(* IEC 61131-3 sources: std_i2980_v2.06_cp053/Source/IMM/ieccontrol/AutoCalibration1 (part 5) *)

@F

@Trans @RT(9)TResetBwd @F @T @F @F @T @T @TL(2)
TRUE

@RT(9)TResetBwd @F
@Goto @RT(7)S_RESET @F @F

@Step @RT(23)S_CHECK_ALARMS_RETRYBWD @F @F @F @F @RT(0) @F
@AcbCont @RT(7)unnamed @F 0

@AltBranch @RT(3)alt @F 2
@TransSeq @RT(4)tseq @F 1
@Trans @RT(9)TRetryBwd @F @T @F @F @T @T @TL(2)
S_CHECK_ALARMS_RETRYBWD.T > T#1s

@RT(9)TRetryBwd @F

@TransSeq @RT(4)tseq @F 2
@Trans @RT(14)TStopIdentBwd4 @F @T @F @F @T @F @TL(2)
sv_iPendingAlarms <> 0

@RT(14)TStopIdentBwd4 @F
@Goto @RT(13)S_StopMoveFwd @F @F

@Goto @RT(11)S_CALIB_BWD @F @F

@Step @RT(12)S_MoveEndBwd @F @F @F @F @RT(0) @F
@AcbCont @RT(7)unnamed @F 3
@Acb @RT(11)AMoveEndBwd @F @T @RT(1)P @RT(0) @F @F @T @TL(27)
bMoveBwdDone := FALSE;

IF mActMovement^.bPositionIncreasingFwd THEN
   mActMovement^.prIdentPosition^ := mrBwdStopPosition;
ELSE
   mActMovement^.prIdentPosition^ := mActMovement^.prStroke^ - mrBwdStopPosition;
END_IF;
mActMovement^.prStopRamp^ := 1.0e10;
mActMovement^.pConstBwdVis^.Pressure.Output.rRamp := MAX(1.0e20,mActMovement^.pConstBwdVis^.Pressure.Output.rRamp);
mActMovement^.pConstBwdVis^.Pressure.rMinOutput := 0.1 * rMaxPressureLimit;
sv_EjectorIdentMinMovement.pConstBwdVis^.Pressure.Output.rRamp := MAX(1.0e10, sv_EjectorIdentMinMovement.pConstBwdVis^.Pressure.Output.rRamp);
sv_EjectorIdentMinMovement.pConstBwdVis^.Pressure.rMinOutput := 0.1 * sv_EjectorIdentMinMovement.prMaxPressureBwd^;

mActMovement^.pbMoveIdent^ := TRUE;

evStartRequestData.DeviceId := mActMovement^.DeviceId;
evStartRequestData.MoveDir := cMoveBwd;
IF mActMovement^.MoveId > cMoveNone THEN
   evStartRequestData.MoveId := cMoveDecompAftPlast;
ELSE
   evStartRequestData.MoveId := cMoveBwd;
END_IF;
miErrorNo := cIdentSpeedMaxEnd;

SET_EVENT(evStartRequest, evStartRequestData);

@F
@Acb @RT(21)ACheckMoveEndBwdReady @F @T @RT(1)N @RT(0) @F @F @T @TL(5)
fbCheckReady(DeviceId := evStartRequestData.DeviceId);
IF fbCheckReady.bReady THEN
   bMoveBwdDone := TRUE;
END_IF;

@F
@Acb @RT(16)AMoveEndBwdReady @F @T @RT(2)P0 @RT(0) @F @F @T @TL(2)
aStopMovementBwd();

@F

@AltBranch @RT(3)alt @F 2
@TransSeq @RT(4)tseq @F 1
@Trans @RT(15)TMoveEndBwdDone @F @T @F @F @T @T @TL(2)
bMoveBwdDone

@RT(15)TMoveEndBwdDone @F

@TransSeq @RT(4)tseq @F 4
@Trans @RT(15)TStopMoveEndBwd @F @T @F @F @T @F @TL(4)
sv_GlobalIdentMaxSpeedStatus.Status = tnCalibState_Aborted OR
sv_GlobalIdentMaxSpeedStatus.Status = tnCalibState_None
OR sv_iPendingAlarms <> 0

@RT(15)TStopMoveEndBwd @F
@Step @RT(16)S_StopMoveEndBwd @F @F @F @F @RT(0) @F
@AcbCont @RT(7)unnamed @F 1
@Acb @RT(15)AStopMoveEndBwd @F @T @RT(1)P @RT(0) @F @F @T @TL(2)
aStopMovementError(sMovementName := CONCAT(sMoveName, ' max ident Bwd to end position'));

@F

@Trans @RT(16)TResetMoveEndBwd @F @T @F @F @T @F @TL(2)
TRUE

@RT(16)TResetMoveEndBwd @F
@Goto @RT(7)S_RESET @F @F

@Step @RT(6)S_Done @F @F @F @F @RT(0) @F
@AcbCont @RT(7)unnamed @F 1
@Acb @RT(5)ADone @F @T @RT(1)P @RT(0) @F @F @T @TL(6)
mActMovement^.Status := tnCalibState_Done;
sv_GlobalIdentMaxSpeedStatus.Status := tnCalibState_Done;

mActMovement^.prVelocityFwd^ := rSpeedLimitFwd;
mActMovement^.prVelocityBwd^ := rSpeedLimitBwd;

@F

@Trans @RT(5)TDone @F @T @F @F @T @T @TL(2)
TRUE

@RT(5)TDone @F
@Goto @RT(7)S_RESET @F @F
@END_SfcData
@SaActions 0
@SaTrans 0
@SaExits 0
@END_SfcBody

@@@BEG_Comment@@@
@TL(0)

@@@END_Comment@@@

@BEG_Body
@TL(35)
//stop all calibrations
// TEST
IF sv_GlobalIdentMaxSpeedStatus.Command = tnCalibCommand_Stop THEN
    sv_GlobalIdentMaxSpeedStatus.bStart := FALSE;
END_IF;
//
IF sv_GlobalIdentMaxSpeedStatus.Command = tnCalibCommand_Stop OR (NOT sv_GlobalIdentMaxSpeedStatus.bStart) THEN
    FOR i:= 1 TO cCalibMovements DO
        IF CHECK_REF(sv_GlobalIdentMaxSpeedStatus.pMovements[i]^) THEN
            IF sv_GlobalIdentMaxSpeedStatus.pMovements[i]^.Status = tnCalibState_Running OR
               sv_GlobalIdentMaxSpeedStatus.pMovements[i]^.bRedo THEN
                sv_GlobalIdentMaxSpeedStatus.pMovements[i]^.Status := tnCalibState_Aborted;
                sv_GlobalIdentMaxSpeedStatus.pMovements[i]^.bRedo := FALSE;//FIXME: check if needed
                sv_GlobalIdentMaxSpeedStatus.Status := tnCalibState_Aborted;
                EXIT;
            END_IF;
        END_IF;
    END_FOR;
    IF (sv_GlobalIdentMaxSpeedStatus.Command = tnCalibCommand_Stop) THEN
       IF (sv_GlobalIdentMaxSpeedStatus.Status <> tnCalibState_Aborted) THEN
          sv_GlobalIdentMaxSpeedStatus.Status := tnCalibState_None;
       END_IF;

    END_IF;
ELSIF (sv_GlobalIdentMaxSpeedStatus.Command = tnCalibCommand_Start) OR (sv_GlobalIdentMaxSpeedStatus.bStart) THEN
    IF sv_OperationMode = nSetup THEN
        mbUseSingleMovement := FALSE;
        START_PROCESS_ALGORITHM(paMaxCalibSequence);
    ELSE
        sv_GlobalIdentMaxSpeedStatus.bStart := FALSE;
        SET_ALARM(erSetupModeRequiredForCalib);
    END_IF;
END_IF;
sv_GlobalIdentMaxSpeedStatus.Command := tnCalibCommand_None;

@END_Body

@@@BEG_Comment@@@
@TL(0)

@@@END_Comment@@@

@BEG_SfcBody
18 18 17

@BEG_SfcData 2
@StepSeq @RT(4)sseq @F 15
@Step @RT(7)S_RESET @F @F @T @F @RT(0) @F
@AcbCont @RT(7)unnamed @F 3
@Acb @RT(6)AReset @F @T @RT(1)P @RT(0) @F @F @T @TL(2)
sv_bAutoIdentRunning := FALSE;

@F
@Acb @RT(14)AStopMovements @F @T @RT(1)N @RT(0) @F @F @T @TL(12)
(* stop all identification movements *)
FOR i:= 1 TO cCalibMovements DO
    IF CHECK_REF(sv_GlobalIdentMaxSpeedStatus.pMovements[i]^) THEN
        IF sv_GlobalIdentMaxSpeedStatus.pMovements[i]^.Status = tnCalibState_Running OR
           sv_GlobalIdentMaxSpeedStatus.pMovements[i]^.bRedo THEN
            sv_GlobalIdentMaxSpeedStatus.pMovements[i]^.Status := tnCalibState_Aborted;
            sv_GlobalIdentMaxSpeedStatus.pMovements[i]^.bRedo := FALSE;//FIXME: check if needed
            EXIT;
        END_IF;
    END_IF;
END_FOR;

@F
@Acb @RT(9)AStopSelf @F @T @RT(1)P @RT(0) @F @F @T @TL(3)
sv_GlobalIdentMaxSpeedStatus.bStart := FALSE;
STOP_PROCESS_ALGORITHM();

@F

@Trans @RT(7)Trans50 @F @T @F @F @T @T @TL(2)
TRUE

@RT(7)Trans50 @F
@Step @RT(6)S_INIT @F @T @F @F @RT(0) @F
@AcbCont @RT(7)unnamed @F 2
@Acb @RT(11)ASortCalibs @F @T @RT(1)P @RT(0) @F @F @T @TL(24)
sv_GlobalIdentMaxSpeedStatus.Status := tnCalibState_Running;
miErrorNo := 0;

tmpMovements := sv_GlobalIdentMaxSpeedStatus.pMovements;

(* get number of movements *)
FOR i:= 1 TO cCalibMovements DO
    IF NOT CHECK_REF(tmpMovements[i]^)  THEN
        EXIT;
    END_IF;
END_FOR;
iMaxMovements := i -1;

(* sort them by iOrder *)
FOR i := 1 TO iMaxMovements -1 DO
    FOR j := 1 TO iMaxMovements - 1 - i +1 DO
        IF tmpMovements[j]^.iOrder > tmpMovements[j + 1]^.iOrder THEN
            tmpM := tmpMovements[j];
            tmpMovements[j] := tmpMovements[j + 1];
            tmpMovements[j + 1] := tmpM;
        END_IF;
    END_FOR;
END_FOR;

@F
@Acb @RT(9)Action108 @F @T @RT(1)P @RT(0) @F @F @T @TL(3)
mCalibCounter := 0;
sv_GlobalIdentMaxSpeedStatus.iCurrentStep := mCalibCounter;

@F

@AltBranch @RT(3)alt @F 2
@TransSeq @RT(4)tseq @F 1
@Trans @RT(7)Trans80 @F @T @F @F @T @T @TL(3)
NOT sv_bCoresActive AND
sv_iPendingAlarms = 0

@RT(7)Trans80 @T @TL(5)
Comment : Start with moving ejector and
mold in backward position, check if any failure
occured.
After that start the calibration cycle, if no alarm is
pending

@TransSeq @RT(4)tseq @F 4
@Trans @RT(7)Trans87 @F @T @F @F @T @F @TL(3)
sv_bCoresActive OR
sv_iPendingAlarms > 0

@RT(7)Trans87 @F
@Step @RT(6)Step74 @F @F @F @F @RT(0) @F
@AcbCont @RT(7)unnamed @F 1
@Acb @RT(14)AAnyCoreActive @F @F @RT(1)N @RT(0) @F @F @F @F

@Trans @RT(7)Trans88 @F @T @F @F @T @T @TL(3)
TRUE

@RT(7)Trans88 @F
@Goto @RT(7)S_RESET @F @F

@Step @RT(6)Step19 @F @F @F @F @RT(0) @F
@AcbCont @RT(7)unnamed @F 1
@Acb @RT(12)ASignalStart @F @T @RT(1)P @RT(0) @F @F @T @TL(2)
sv_bAutoIdentRunning := TRUE;

@F

@Trans @RT(7)Trans18 @F @T @F @F @T @T @TL(2)
TRUE

@RT(7)Trans18 @F
@Step @RT(17)S_MoveEjectorBack @F @F @F @F @RT(0) @F
@AcbCont @RT(7)unnamed @F 3
@Acb @RT(12)AEjectorBack @F @F @RT(1)P @RT(0) @F @F @F @F
@Acb @RT(9)Action116 @F @T @RT(1)N @RT(0) @F @F @T @TL(2)
fbCheckReady(DeviceId := DeviceIdEjector)

@F
@Acb @RT(17)AResetEjectorBack @F @T @RT(2)P0 @RT(0) @F @F @T @TL(7)
miErrorNo := 0;
sv_EjectorIdentMaxMovement.prIdentPosition^ := 0.0;
sv_EjectorIdentMaxMovement.prStopRamp^ := 0.0;
sv_EjectorIdentMaxMovement.pbMoveIdent^ := FALSE;
sv_EjectorIdentMaxMovement.pConstBwdVis^ := ConstBwdVis;

@F

@AltBranch @RT(3)alt @F 2
@TransSeq @RT(4)tseq @F 1
@Trans @RT(7)Trans72 @F @T @F @F @T @T @TL(3)
fbCheckReady.bReady AND
sv_iPendingAlarms = 0

@RT(7)Trans72 @F

@TransSeq @RT(4)tseq @F 4
@Trans @RT(7)Trans83 @F @T @F @F @T @F @TL(4)
sv_GlobalIdentMaxSpeedStatus.Status = tnCalibState_Aborted OR
sv_GlobalIdentMaxSpeedStatus.Status = tnCalibState_None
OR sv_iPendingAlarms <> 0

@RT(7)Trans83 @F
@Step @RT(13)S_StopEjector @F @F @F @F @RT(0) @F
@AcbCont @RT(7)unnamed @F 1
@Acb @RT(16)AStopEjeMovement @F @F @RT(1)P @RT(0) @F @F @F @F

@Trans @RT(7)Trans84 @F @T @F @F @T @T @TL(3)
TRUE

@RT(7)Trans84 @F
@Goto @RT(7)S_RESET @F @F

@Step @RT(14)S_MoveMoldBack @F @F @F @F @RT(0) @F
@AcbCont @RT(7)unnamed @F 3
@Acb @RT(9)AMoldBack @F @F @RT(1)P @RT(0) @F @F @F @F
@Acb @RT(9)Action118 @F @T @RT(1)N @RT(0) @F @F @T @TL(2)
fbCheckReady(DeviceId := DeviceIdMold)

@F
@Acb @RT(14)AResetMoldBack @F @T @RT(2)P0 @RT(0) @F @F @T @TL(7)
miErrorNo := 0;
sv_MoldIdentMaxMovement.prIdentPosition^ := 0.0;
sv_MoldIdentMaxMovement.prStopRamp^ := 0.0;
sv_MoldIdentMaxMovement.pbMoveIdent^ := FALSE;
sv_MoldIdentMaxMovement.pConstBwdVis^ := ConstBwdVis;

@F

@AltBranch @RT(3)alt @F 2
@TransSeq @RT(4)tseq @F 1
@Trans @RT(7)Trans81 @F @T @F @F @T @T @TL(3)
fbCheckReady.bReady AND
sv_iPendingAlarms = 0

@RT(7)Trans81 @F

@TransSeq @RT(4)tseq @F 4
@Trans @RT(7)Trans85 @F @T @F @F @T @F @TL(4)
sv_GlobalIdentMaxSpeedStatus.Status = tnCalibState_Aborted OR
sv_GlobalIdentMaxSpeedStatus.Status = tnCalibState_None
OR sv_iPendingAlarms <> 0

@RT(7)Trans85 @F
@Step @RT(10)S_StopMold @F @F @F @F @RT(0) @F
@AcbCont @RT(7)unnamed @F 1
@Acb @RT(17)AStopMoldMovement @F @F @RT(1)P @RT(0) @F @F @F @F

@Trans @RT(7)Trans86 @F @T @F @F @T @T @TL(2)
TRUE

@RT(7)Trans86 @F
@Goto @RT(7)S_RESET @F @F

@Step @RT(14)S_CALIB_SINGLE @F @F @T @F @RT(0) @F
@AcbCont @RT(7)unnamed @F 1
@Acb @RT(19)AStartMovementStart @F @T @RT(1)P @RT(0) @F @F @T @TL(5)
IF mCalibCounter < iMaxMovements THEN
   mCalibCounter := mCalibCounter +1;
   tmpMovements[mCalibCounter]^.bRedo := TRUE;
END_IF;

@F

@AltBranch @RT(3)alt @F 2
@TransSeq @RT(4)tseq @F 1
@Trans @RT(18)TCheckActMoveReady @F @T @F @F @T @T @TL(4)
tmpMovements[mCalibCounter]^.bRedo = FALSE AND
NOT(sv_GlobalIdentMaxSpeedStatus.Status = tnCalibState_Aborted OR
    sv_GlobalIdentMaxSpeedStatus.Status = tnCalibState_Error)

@RT(18)TCheckActMoveReady @F

@TransSeq @RT(4)tseq @F 2
@Trans @RT(11)TCheckError @F @T @F @F @T @F @TL(4)
sv_GlobalIdentMaxSpeedStatus.Status = tnCalibState_Aborted OR
sv_GlobalIdentMaxSpeedStatus.Status = tnCalibState_Error OR
iMaxMovements = 0

@RT(11)TCheckError @F
@Goto @RT(7)S_RESET @F @F

@Step @RT(11)S_CHECKNEXT @F @F @F @F @RT(0) @F
@AcbCont @RT(7)unnamed @F 0

@AltBranch @RT(3)alt @F 2
@TransSeq @RT(4)tseq @F 1
@Trans @RT(9)TNextUnit @F @T @F @F @T @T @TL(2)
mCalibCounter < iMaxMovements

@RT(9)TNextUnit @F

@TransSeq @RT(4)tseq @F 4
@Trans @RT(10)TStopIdent @F @T @F @F @T @T @TL(2)
mCalibCounter >= iMaxMovements

@RT(10)TStopIdent @F
@Step @RT(11)S_StopIdent @F @F @F @F @RT(0) @F
@AcbCont @RT(7)unnamed @F 1
@Acb @RT(10)AStopIdent @F @T @RT(1)P @RT(0) @F @F @T @TL(2)
sv_GlobalIdentMaxSpeedStatus.Status := tnCalibState_Done;

@F

@Trans @RT(6)TReset @F @T @F @F @T @T @TL(2)
TRUE

@RT(6)TReset @F
@Goto @RT(7)S_RESET @F @F

@Goto @RT(14)S_CALIB_SINGLE @F @F
@END_SfcData
@SaActions 5
@SaText @RT(12)AEjectorBack 1 @TL(20)
miErrorNo := cIdentSpeedMaxSequence;

IF sv_EjectorIdentMaxMovement.bPositionIncreasingFwd THEN
   sv_EjectorIdentMaxMovement.prIdentPosition^ := mrBwdStopPosition;
ELSE
   sv_EjectorIdentMaxMovement.prIdentPosition^ := sv_EjectorIdentMaxMovement.prStroke^ - mrBwdStopPosition;
END_IF;
sv_EjectorIdentMaxMovement.prStopRamp^ := 1.0e10;
ConstBwdVis := sv_EjectorIdentMaxMovement.pConstBwdVis^;
sv_EjectorIdentMaxMovement.pConstBwdVis^.Pressure.Output.rRamp := MAX(1.0e10, sv_EjectorIdentMaxMovement.pConstBwdVis^.Pressure.Output.rRamp);
sv_EjectorIdentMaxMovement.pConstBwdVis^.Pressure.rMinOutput := 0.1 * sv_EjectorIdentMaxMovement.prMaxPressureBwd^;
sv_EjectorIdentMaxMovement.pbMoveIdent^ := TRUE;

evStartRequestData.DeviceId := DeviceIdEjector;
evStartRequestData.MoveDir := cMoveBwd;
evStartRequestData.MoveId := cMoveBwd;
SET_EVENT(evStartRequest, evStartRequestData);

@SaText @RT(9)AMoldBack 1 @TL(19)
miErrorNo := cIdentSpeedMaxSequence;

IF sv_MoldIdentMaxMovement.bPositionIncreasingFwd THEN
   sv_MoldIdentMaxMovement.prIdentPosition^ := mrBwdStopPosition;
ELSE
   sv_MoldIdentMaxMovement.prIdentPosition^ := sv_MoldIdentMaxMovement.prStroke^ - mrBwdStopPosition;
END_IF;
sv_MoldIdentMaxMovement.prStopRamp^ := 1.0e10;
ConstBwdVis := sv_MoldIdentMaxMovement.pConstBwdVis^;
sv_MoldIdentMaxMovement.pConstBwdVis^.Pressure.Output.rRamp := MAX(1.0e10, sv_MoldIdentMaxMovement.pConstBwdVis^.Pressure.Output.rRamp);
sv_MoldIdentMaxMovement.pConstBwdVis^.Pressure.rMinOutput := 0.1 * sv_MoldIdentMaxMovement.prMaxPressureBwd^;
sv_MoldIdentMaxMovement.pbMoveIdent^ := TRUE;

evStartRequestData.DeviceId := DeviceIdMold;
evStartRequestData.MoveDir := cMoveBwd;
evStartRequestData.MoveId := cMoveBwd;
SET_EVENT(evStartRequest, evStartRequestData);

@SaText @RT(16)AStopEjeMovement 1 @TL(9)
evStopRequestData.DeviceId := DeviceIdEjector;
evStopRequestData.MoveDir := cMoveBwd;
evStopRequestData.MoveId := cMoveBwd;
SET_EVENT(evStopRequest, evStopRequestData);
IF sv_GlobalIdentMaxSpeedStatus.Status <> tnCalibState_None THEN
    sv_GlobalIdentMaxSpeedStatus.Status := tnCalibState_Aborted;
END_IF;

@SaText @RT(17)AStopMoldMovement 1 @TL(9)
evStopRequestData.DeviceId := DeviceIdMold;
evStopRequestData.MoveDir := cMoveBwd;
evStopRequestData.MoveId := cMoveBwd;
SET_EVENT(evStopRequest, evStopRequestData);
IF sv_GlobalIdentMaxSpeedStatus.Status <> tnCalibState_None THEN
    sv_GlobalIdentMaxSpeedStatus.Status := tnCalibState_Aborted;
END_IF;

@SaText @RT(14)AAnyCoreActive 1 @TL(6)
IF sv_bCoresActive THEN
   SET_ALARM(erCalibCoresActive);
END_IF;
sv_GlobalIdentMaxSpeedStatus.Status := tnCalibState_Aborted;

@SaTrans 0
@SaExits 1
@SaExit @SaText @RT(14)E_NotSetupMode 1 @TL(2)
sv_OperationMode <> nSetup

@RT(7)S_RESET @RT(1)1 @F @F @SaSfc @RT(14)E_NotSetupMode 5 @RT(5)DUMMY
@BEG_SfcData 2
@ExitSeq @RT(4)sseq @F 3
@Step @RT(8)unnamed1 @F @T @F @F @RT(0) @F
@AcbCont @RT(7)unnamed @F 0

@Trans @RT(8)unnamed3 @F @T @F @F @T @T @TL(2)

@RT(8)unnamed3 @F
@Goto @RT(9)unlabeled @F @F
@END_SfcData

@END_SfcBody

@@@BEG_Comment@@@
@TL(2)
Coordinate sequential start of auto calib cycle
starts one auto calib movement after the other
@@@END_Comment@@@

@BEG_Body
@TL(7)
IF (rStep > 0.0) THEN
   rRealValue := (0.999 + rActNumber / rStep);
   rRoundedNumber := DINT_TO_REAL(TRUNC_TO_DINT(rRealValue)) * rStep;
ELSE
   rRoundedNumber := rActNumber;
END_IF;

@END_Body

@@@BEG_Comment@@@
@TL(0)

@@@END_Comment@@@

@BEG_Body
@TL(39)
IF bStart THEN
   rMaxRefSpeed := rMaxSpeedLimit;
   rMinRefSpeed := 0.0;
END_IF;
IF (bUnstable OR bTimeOut) THEN
   // increase speed
   IF (rActRefSpeed >= rMFactorMaxMinLimit * rMaxSpeedLimit) THEN
      bMinDetected := TRUE;
      rMinSpeed := rActRefSpeed;
      RETURN;
   END_IF;
   rMinRefSpeed := rActRefSpeed;
   bMinDetected := FALSE;
  IF (rMaxRefSpeed - rMinRefSpeed) < (0.0025 * rMaxSpeedLimit) THEN
  // difference to low to maximum - stop or increase maximum?
      bMinDetected := TRUE;
      rMinSpeed := rMaxRefSpeed;
   ELSIF (rMaxRefSpeed < rMaxSpeedLimit) AND (rMinRefSpeed > 0.0) THEN
      rRefSpeed := 0.5 * (rMaxRefSpeed + rMinRefSpeed);
      bMinDetected := FALSE;
   ELSE
      rRefSpeed := rActRefSpeed + 0.01 * rMaxSpeedLimit;
      IF (rRefSpeed >= rMaxSpeedLimit) THEN
         bMinDetected := TRUE;
         rMinSpeed := rMaxSpeedLimit;
      END_IF;
   END_IF;
ELSE
   // reduce speed
   rMaxRefSpeed := rActRefSpeed;
   IF (rMaxRefSpeed - rMinRefSpeed) < (0.0025 * rMaxSpeedLimit) THEN
      bMinDetected := TRUE;
      rMinSpeed := rActRefSpeed;
   ELSE
      bMinDetected := FALSE;
      rRefSpeed := 0.5 * (rMaxRefSpeed + rMinRefSpeed);
   END_IF;
END_IF;

@END_Body

@@@BEG_Comment@@@
@TL(0)

@@@END_Comment@@@

@BEG_Body
@TL(26)
bIdentActive := FALSE;
FOR i:= 1 TO cCalibMovements DO
   IF CHECK_REF(sv_GlobalIdentMinSpeedStatus.pMovements[i]^) THEN
      IF sv_GlobalIdentMinSpeedStatus.pMovements[i]^.bRedo THEN
         mActMovement := sv_GlobalIdentMinSpeedStatus.pMovements[i];
         bIdentActive := TRUE;
         sv_GlobalIdentMinSpeedStatus.iCurrentStep :=  i;
         mCalibCounter := i;
         IF sv_OperationMode = nSetup THEN
            mbUseSingleMovement := TRUE;
            START_PROCESS_ALGORITHM(paMinSingleMovement);
         ELSE
            sv_GlobalIdentMinSpeedStatus.pMovements[i]^.bRedo := FALSE;
            SET_ALARM(erSetupModeRequiredForCalib);
         END_IF;
         EXIT;
      END_IF;
   END_IF;
END_FOR;
IF ((NOT bIdentActive) AND (sv_GlobalIdentMinSpeedStatus.Status = tnCalibState_Running)) THEN
   sv_GlobalIdentMinSpeedStatus.Status := tnCalibState_Done;
END_IF;

STOP_PROCESS_ALGORITHM();

@END_Body

@@@BEG_Comment@@@
@TL(0)

@@@END_Comment@@@

@BEG_Body
@TL(4)

START_PROCESS_ALGORITHM(paRedoMin);

@END_Body

@@@BEG_Comment@@@
@TL(0)

@@@END_Comment@@@

@BEG_SfcBody
44 51 50

@BEG_SfcData 2
@StepSeq @RT(4)sseq @F 39
@Step @RT(7)S_RESET @F @F @T @F @RT(0) @F
@AcbCont @RT(7)unnamed @F 0

@Trans @RT(7)Trans47 @F @T @F @F @T @T @TL(2)
mbLogFileSaved

@RT(7)Trans47 @F
@Step @RT(6)S_STOP @F @F @F @F @RT(0) @F
@AcbCont @RT(7)unnamed @F 1
@Acb @RT(9)AStopSelf @F @T @RT(1)P @RT(0) @F @F @T @TL(18)
IF (sv_GlobalIdentMinSpeedStatus.Status = tnCalibState_Aborted) THEN
   mActMovement^.prVelocityFwd^ := rSpeedLimitFwd;
   mActMovement^.prVelocityBwd^ := rSpeedLimitBwd;
END_IF;
sv_GlobalIdentMinSpeedStatus.Command := tnCalibCommand_None;
sv_bAutoIdentRunning := FALSE;
mActMovement^.bRedo := FALSE;
mActMovement^.pdMaxMoveTimeFwd^ := dMaxMoveTimeSaveFwd;
mActMovement^.pdMaxMoveTimeBwd^ := dMaxMoveTimeSaveBwd;
mActMovement^.prStopRamp^ := 0.0;
mActMovement^.pConstFwdVis^ := ConstVisFwd;
mActMovement^.pConstBwdVis^ := ConstVisBwd;

//release memory
abSpeedMeasure.aEnd();

STOP_PROCESS_ALGORITHM();

@F

@Trans @RT(8)TRestart @F @T @F @F @T @T @TL(2)
TRUE

@RT(8)TRestart @F
@Step @RT(6)S_INIT @F @T @F @F @RT(0) @F
@AcbCont @RT(7)unnamed @F 1
@Acb @RT(7)Action3 @F @T @RT(1)P @RT(0) @F @F @T @TL(38)
miErrorNo := 0;

sv_GlobalIdentMinSpeedStatus.Status := tnCalibState_Running;
mActMovement^.Status := tnCalibState_Running;
sMoveName := mActMovement^.sName;

abSpeedMeasure.aInit();

bMinFwdRetry := FALSE;
bMinBwdRetry := FALSE;

dMaxMoveTimeSaveFwd := mActMovement^.pdMaxMoveTimeFwd^;
dMaxMoveTimeSaveBwd := mActMovement^.pdMaxMoveTimeBwd^;

ConstVisFwd := mActMovement^.pConstFwdVis^;
ConstVisBwd := mActMovement^.pConstBwdVis^;

rSpeedLimitFwd := mActMovement^.prVelocityFwd^;
rSpeedLimitBwd := mActMovement^.prVelocityBwd^;

IF (mActMovement^.rMaxPositionLimitFactor > mActMovement^.rMinPositionLimitFactor) AND
   (mActMovement^.rMinPositionLimitFactor > 0.0) AND (mActMovement^.rMaxPositionLimitFactor < 1.0) THEN
   mrMaxPositionFactor := mActMovement^.rMaxPositionLimitFactor;
   mrMinPositionFactor := mActMovement^.rMinPositionLimitFactor;
ELSE // use deafult values
   mrMaxPositionFactor := 0.8;
   mrMinPositionFactor := 0.2;
END_IF;

rMaxPressureFwd := 0.0;
rMaxPressureBwd := 0.0;
mprActPressure := sv_PumpData[mActMovement^.DeviceId.IndexId].prActSysPressure;
IF CHECK_REF(mprActPressure^) THEN
   mbprActPressureLinked := TRUE;
ELSE
   mbprActPressureLinked := FALSE;
END_IF;

@F

@Trans @RT(13)TMoveStartBwd @F @T @F @F @T @T @TL(3)
TRUE

@RT(13)TMoveStartBwd @F
@Step @RT(14)S_MoveStartBwd @F @F @F @F @RT(0) @F
@AcbCont @RT(7)unnamed @F 3
@Acb @RT(13)AMoveStartBwd @F @T @RT(1)P @RT(0) @F @F @T @TL(4)
bMoveBwdDone := FALSE;
miErrorNo := cIdentSpeedMinBwdInit;
aStartMovementBwd();

@F
@Acb @RT(23)ACheckMoveStartBwdReady @F @T @RT(1)N @RT(0) @F @F @T @TL(5)
fbCheckReady(DeviceId := evStartRequestData.DeviceId);
IF fbCheckReady.bReady THEN
   bMoveBwdDone := TRUE;
END_IF;

@F
@Acb @RT(18)AMoveStartBwdReady @F @T @RT(2)P0 @RT(0) @F @F @T @TL(5)
aStopMovementBwd();

@F

@AltBranch @RT(3)alt @F 2
@TransSeq @RT(4)tseq @F 1
@Trans @RT(8)TInitBwd @F @T @F @F @T @T @TL(2)
bMoveBwdDone

@RT(8)TInitBwd @F

@TransSeq @RT(4)tseq @F 4
@Trans @RT(17)TStopMoveStartBwd @F @T @F @F @T @F @TL(5)
sv_GlobalIdentMinSpeedStatus.Status = tnCalibState_Aborted OR
sv_GlobalIdentMinSpeedStatus.Status = tnCalibState_None
OR sv_iPendingAlarms <> 0
OR mActMovement^.bRedo = FALSE

@RT(17)TStopMoveStartBwd @F
@Step @RT(18)S_StopMoveStartBwd @F @F @T @F @RT(0) @F
@AcbCont @RT(7)unnamed @F 1
@Acb @RT(22)AStopMoveErrorStartBwd @F @T @RT(1)P @RT(0) @F @F @T @TL(2)
aStopMovementError(sMovementName := CONCAT(sMoveName, ' min ident Fwd: Bwd to initial position'));

@F

@Trans @RT(6)TReset @F @T @F @F @T @F @TL(2)
TRUE

@RT(6)TReset @F
@Goto @RT(7)S_RESET @F @F

@Step @RT(22)S_CHECK_ALARMS_INITBWD @F @F @F @F @RT(0) @F
@AcbCont @RT(7)unnamed @F 0

@AltBranch @RT(3)alt @F 2
@TransSeq @RT(4)tseq @F 1
@Trans @RT(11)TStartIdent @F @T @F @F @T @T @TL(2)
S_CHECK_ALARMS_INITBWD.T > T#100ms

@RT(11)TStartIdent @F

@TransSeq @RT(4)tseq @F 2
@Trans @RT(12)TStopInitBwd @F @T @F @F @T @F @TL(2)
sv_iPendingAlarms <> 0

@RT(12)TStopInitBwd @F
@Goto @RT(18)S_StopMoveStartBwd @F @F

@Step @RT(15)S_INITCALIB_FWD @F @F @F @F @RT(0) @F
@AcbCont @RT(7)unnamed @F 1
@Acb @RT(13)aInitIdentFwd @F @T @RT(1)P @RT(0) @F @F @T @TL(26)
iFileCounter := 1;
IF (CHECK_REF(mActMovement^.prSizeFactorFwd^)) THEN
   IF (mActMovement^.prSizeFactorFwd^ > 0.0) THEN
      rVelocitSizeFactor := mActMovement^.prSizeFactorFwd^;
   END_IF;
ELSE
   rVelocitSizeFactor := 1.0;
END_IF;
rRefSpeedLimit := 0.01 * mActMovement^.prVelocityLimitFwd^;
rMaxPressureLimit := mActMovement^.prMaxPressureFwd^;
IF CHECK_REF(mActMovement^.prMaxPressureFwdHydr^) THEN
   rMaxRefPressureLimit := mActMovement^.prMaxPressureFwdHydr^;
   IF (rMaxRefPressureLimit > 0.0) THEN
      rPressureFactorFwd := rMaxPressureLimit / rMaxRefPressureLimit;
   ELSE
      rPressureFactorFwd := 1.0;
   END_IF;
ELSE
   rMaxRefPressureLimit := mActMovement^.prMaxPressureFwd^;
   rPressureFactorFwd := 1.0;
END_IF;

aCalcMinSpeedOutput.bStart := TRUE;

dummy := Print('Calib min output %s Fwd started', sMoveName);

@F

@Trans @RT(7)TDelay1 @F @T @F @F @T @T @TL(2)
S_INITCALIB_FWD.T>T#100ms

@RT(7)TDelay1 @F
@Step @RT(11)S_CALIB_FWD @F @F @T @F @RT(0) @F
@AcbCont @RT(7)unnamed @F 4
@Acb @RT(8)ADoCalib @F @T @RT(1)P @RT(0) @F @F @T @TL(67)
// save actual settings
mActMovement^.pConstFwdVis^.Velocity.Output.rOutputValue := rRefSpeedLimit * rVelocitSizeFactor;
mActMovement^.pConstFwdVis^.Velocity.rMinOutput := 0.0;
mActMovement^.pConstFwdVis^.Pressure.Output.rOutputValue := MAX(mActMovement^.pConstFwdVis^.Pressure.Output.rOutputValue, rMaxPressureLimit);
mActMovement^.pConstFwdVis^.Pressure.Output.rRamp := MAX(1.0e10, ConstVisFwd.Pressure.Output.rRamp);
IF mActMovement^.bPositionIncreasingFwd THEN
   mActMovement^.prIdentPosition^ := mActMovement^.prStroke^ * mrMaxPositionFactor;
   mrMinLimitPosition := rStartFactor * mActMovement^.prIdentPosition^ + (1.0 - rStartFactor) * mActMovement^.prPosition^;
   IF (mActMovement^.prIdentPosition^ - mActMovement^.prPosition^) > 0.0 THEN
      rMinStopRamp := rMinStrokeFactor * rRefSpeedLimit  * rRefSpeedLimit / ABS(mActMovement^.prIdentPosition^ - mActMovement^.prPosition^);
   ELSE
      rMinStopRamp := 0.0;
   END_IF;
   mActMovement^.prStopRamp^ := MAX(mActMovement^.pConstFwdVis^.Velocity.Output.rRamp, rMinStopRamp);
   mrMaxLimitPosition := mActMovement^.prIdentPosition^ - 0.5 * rRefSpeedLimit  * rRefSpeedLimit / mActMovement^.prStopRamp^;
ELSE
   mActMovement^.prIdentPosition^ := mActMovement^.prStroke^ * mrMinPositionFactor;
   mrMaxLimitPosition := (1.0 - rStartFactor) * mActMovement^.prPosition^ + rStartFactor * mActMovement^.prIdentPosition^;
   IF (mActMovement^.prPosition^ - mActMovement^.prIdentPosition^) > 0.0 THEN
      rMinStopRamp := rMinStrokeFactor * rRefSpeedLimit  * rRefSpeedLimit / ABS(mActMovement^.prIdentPosition^ - mActMovement^.prPosition^);
   ELSE
      rMinStopRamp := 0.0;
   END_IF;
   mActMovement^.prStopRamp^ := MAX(mActMovement^.pConstFwdVis^.Velocity.Output.rRamp, rMinStopRamp);
   mrMinLimitPosition := mActMovement^.prIdentPosition^ + 0.5 * rRefSpeedLimit  * rRefSpeedLimit / mActMovement^.prStopRamp^;
END_IF;
mActMovement^.pbMoveIdent^ := TRUE;
bMoveIdentDone := FALSE;

bMinFwdDetected := FALSE;

mrRefVelocity := rRefSpeedLimit;
mrRefPressure := rMaxRefPressureLimit;

aStartMeasurement();

bStopUnstable := FALSE;
bTimeOut := FALSE;
IF rRefSpeedLimit > 0.0 THEN
   rMoveStrokeTime := mActMovement^.prStroke^ / rRefSpeedLimit;
ELSE
   rMoveStrokeTime := 0.0;
END_IF;
dMaxMoveTime := T#5s + LINT_TO_TIME(REAL_TO_LINT(rMoveStrokeTime*1.0e6));
IF (dMaxMoveTime > dMoveTimeLimit) THEN
   dMaxMoveTime := dMoveTimeLimit;
   bMoveTimeLimited := TRUE;
   rStartPosition := mActMovement^.prPosition^;
   IF (mActMovement^.bPositionIncreasingFwd) THEN
      rMinMovementPosition := rStartPosition + 0.1 * (mrMaxLimitPosition - mrMinLimitPosition);
   ELSE;
      rMinMovementPosition := rStartPosition - 0.1 * (mrMaxLimitPosition - mrMinLimitPosition );
   END_IF;
ELSE
   bMoveTimeLimited := FALSE;
END_IF;
TimeOut(IN := FALSE,
        PT := dMaxMoveTime);
IF (mActMovement^.pdMaxMoveTimeFwd^ < dMaxMoveTime + dMoveTimeOffset) THEN
   mActMovement^.pdMaxMoveTimeFwd^ := dMaxMoveTime + dMoveTimeOffset;
END_IF;
mActMovement^.prVelocityFwd^ := rRefSpeedLimit;

sWriteSpeedLimit := REAL_TO_STRING(rRefSpeedLimit);
dummy := Print('Calib min output: act. min output: %s', sWriteSpeedLimit);
miErrorNo := cIdentSpeedMinFwdIdent;

@F
@Acb @RT(17)AStartMovementFwd @F @T @RT(1)P @RT(0) @F @F @T @TL(10)
evStartRequestData.DeviceId := mActMovement^.DeviceId;
evStartRequestData.MoveDir := cMoveFwd;
IF mActMovement^.MoveId > cMoveNone THEN
   evStartRequestData.MoveId := mActMovement^.MoveId;
ELSE
   evStartRequestData.MoveId := cMoveFwd;
END_IF;
SET_EVENT(evStartRequest, evStartRequestData);

@F
@Acb @RT(25)ACheckActMovementFwdReady @F @T @RT(1)N @RT(0) @F @F @T @TL(26)
fbCheckReady(DeviceId := evStartRequestData.DeviceId);

TimeOut(IN := TRUE);
IF (fbCheckReady.bReady) THEN
   aStopMeasurement();
   aStopMovementFwd();
   bMoveIdentDone := TRUE;
ELSIF (TimeOut.Q) THEN
   aStopMeasurement();
   aStopMovementFwd();
   IF (bMoveTimeLimited) AND
     ((mActMovement^.bPositionIncreasingFwd AND (mActMovement^.prPosition^ > rMinMovementPosition)) OR
      (NOT mActMovement^.bPositionIncreasingFwd AND (mActMovement^.prPosition^ < rMinMovementPosition))) THEN
      bMoveIdentDone := TRUE;
      dummy := Print('Calib min output: max move time reached with act. min output %s', sWriteSpeedLimit);
   ELSE
      bTimeOut := TRUE;
      dummy := Print('Calib min output: timeout with act. min output %s', sWriteSpeedLimit);
   END_IF;
ELSIF (abSpeedMeasure.aMeasure.bSpeedUnStable) THEN
   aStopMeasurement();
   aStopMovementFwd();
   bStopUnstable := TRUE;
   dummy := Print('Calib min output: unstable speed with act. min output %s', sWriteSpeedLimit);
END_IF;

@F
@Acb @RT(16)AStopMovementFwd @F @T @RT(2)P0 @RT(0) @F @F @T @TL(8)
mActMovement^.prStopRamp^ := 0.0;
mActMovement^.pConstFwdVis^ := ConstVisFwd;
mActMovement^.pdMaxMoveTimeFwd^ := dMaxMoveTimeSaveFwd;

TimeOut(IN := FALSE);

@F

@AltBranch @RT(3)alt @F 2
@TransSeq @RT(4)tseq @F 1
@Trans @RT(17)TMoveIdentFwdDone @F @T @F @F @T @T @TL(4)
bMoveIdentDone OR
bTimeOut OR
bStopUnstable

@RT(17)TMoveIdentFwdDone @F

@TransSeq @RT(4)tseq @F 4
@Trans @RT(13)TStopIdentFwd @F @T @F @F @T @F @TL(5)
sv_GlobalIdentMinSpeedStatus.Status = tnCalibState_Aborted OR
sv_GlobalIdentMinSpeedStatus.Status = tnCalibState_None
OR sv_iPendingAlarms <> 0
OR mActMovement^.bRedo = FALSE

@RT(13)TStopIdentFwd @F
@Step @RT(14)S_StopIdentFwd @F @F @T @F @RT(0) @F
@AcbCont @RT(7)unnamed @F 1
@Acb @RT(13)AStopIdentFwd @F @T @RT(1)P @RT(0) @F @F @T @TL(3)
aStopMovementFwd();
aStopMovementError(sMovementName := CONCAT(sMoveName, ' min ident Fwd'));

@F

@Trans @RT(7)TReset1 @F @T @F @F @T @F @TL(2)
TRUE

@RT(7)TReset1 @F
@Goto @RT(7)S_RESET @F @F

@Step @RT(18)S_CHECK_ALARMS_FWD @F @F @F @F @RT(0) @F
@AcbCont @RT(7)unnamed @F 0

@AltBranch @RT(3)alt @F 2
@TransSeq @RT(4)tseq @F 1
@Trans @RT(14)TStartWriteFwd @F @T @F @F @T @T @TL(2)
S_CHECK_ALARMS_FWD.T > T#100ms

@RT(14)TStartWriteFwd @F

@TransSeq @RT(4)tseq @F 2
@Trans @RT(14)TStopIdentFwd2 @F @T @F @F @T @F @TL(2)
sv_iPendingAlarms <> 0

@RT(14)TStopIdentFwd2 @F
@Goto @RT(14)S_StopIdentFwd @F @F

@Step @RT(11)S_WRITE_FWD @F @F @F @F @RT(0) @F
@AcbCont @RT(7)unnamed @F 1
@Acb @RT(9)AWriteFwd @F @T @RT(1)P @RT(0) @F @F @T @TL(14)
abSpeedMeasure.aGetMaxValues(rMaxSpeed => mrMaxVelocity,
                             rMaxPressure => mrMaxPressure,
                             bPressureLimitReached => mbPressureLimitReached,
                             bSpeedLimitReached => mbVelocityLimitReached);
IF mbprActPressureLinked THEN
   rMaxPressureFwd := MAX(rMaxPressureFwd,mrMaxPressure);
   dummy := Print('Calib min output: with act. min output %s max pressure %f needed', sWriteSpeedLimit, mrMaxPressure);
END_IF;
sFileName := CONCAT(sMoveName,"_MINSPEED_FWD_");
aWriteLog(sFileName := sFileName,
          iFileCounter := iFileCounter,
          bDeleteFiles := TRUE);
iFileCounter := iFileCounter + 1;

@F

@AltBranch @RT(3)alt @F 2
@TransSeq @RT(4)tseq @F 1
@Trans @RT(9)TWriteFwd @F @T @F @F @T @T @TL(2)
mbLogFileSaved

@RT(9)TWriteFwd @F

@TransSeq @RT(4)tseq @F 4
@Trans @RT(16)TAbortedWriteFwd @F @T @F @F @T @F @TL(2)
sv_GlobalIdentMinSpeedStatus.Status = tnCalibState_Aborted

@RT(16)TAbortedWriteFwd @F
@Step @RT(17)S_AbortedWriteFwd @F @F @F @F @RT(0) @F
@AcbCont @RT(7)unnamed @F 1
@Acb @RT(22)AStopMoveErrorWriteFwd @F @T @RT(1)P @RT(0) @F @F @T @TL(3)
mActMovement^.Status := tnCalibState_Error;

@F

@Trans @RT(21)TResetAbortedWriteFwd @F @T @F @F @T @F @TL(2)
TRUE

@RT(21)TResetAbortedWriteFwd @F
@Goto @RT(7)S_RESET @F @F

@Step @RT(20)S_CHECK_MINSPEED_FWD @F @F @F @F @RT(0) @F
@AcbCont @RT(7)unnamed @F 1
@Acb @RT(17)ACheckMinSpeedFwd @F @T @RT(1)P @RT(0) @F @F @T @TL(20)
aCalcMinSpeedOutput(rMaxSpeedLimit := mActMovement^.prVelocityLimitFwd^,
                    rActRefSpeed := rRefSpeedLimit,
                    rActMinSpeed := abSpeedMeasure.aGetMaxValues.rMaxSpeed,
                    bUnstable := abSpeedMeasure.aGetMaxValues.bSpeedLimitUnStable,
                    bTimeOut := bTimeOut);
bMinFwdDetected := aCalcMinSpeedOutput.bMinDetected;
IF (bMinFwdDetected) THEN
   rSpeedLimitFwd := aCalcMinSpeedOutput.rMinSpeed;
   dummy := Print('Calib min output %s Fwd finished: min output fwd = %f$N', sMoveName, rSpeedLimitFwd);
ELSE
   bMinFwdRetry := TRUE;
   rRefSpeedLimit := aCalcMinSpeedOutput.rRefSpeed;
   aCalcMinSpeedOutput.bStart := FALSE;
END_IF;

mActMovement^.pConstFwdVis^ := ConstVisFwd;
mActMovement^.prVelocityFwd^ := rSpeedLimitFwd;
mActMovement^.pdMaxMoveTimeFwd^ := dMaxMoveTimeSaveFwd;

@F

@AltBranch @RT(3)alt @F 2
@TransSeq @RT(4)tseq @F 3
@Trans @RT(15)TMinFwdDetected @F @T @F @F @T @T @TL(2)
bMinFwdDetected

@RT(15)TMinFwdDetected @F
@Step @RT(21)S_ReadyMinFwdDetected @F @F @F @F @RT(0) @F
@AcbCont @RT(7)unnamed @F 1
@Acb @RT(20)AReadyMinFwdDetected @F @T @RT(1)N @RT(0) @F @F @T @TL(2)
fbCheckReady(DeviceId := mActMovement^.DeviceId);

@F

@Trans @RT(20)TReadyMinFwdDetected @F @T @F @F @T @T @TL(2)
fbCheckReady.bReady

@RT(7)Trans49 @F

@TransSeq @RT(4)tseq @F 8
@Trans @RT(7)Trans15 @F @T @F @F @T @T @TL(2)
bMinFwdRetry

@RT(7)Trans15 @F
@Step @RT(18)S_ReadyMinFwdRetry @F @F @F @F @RT(0) @F
@AcbCont @RT(7)unnamed @F 1
@Acb @RT(17)AReadyMinFwdRetry @F @T @RT(1)N @RT(0) @F @F @T @TL(2)
fbCheckReady(DeviceId := mActMovement^.DeviceId);

@F

@Trans @RT(17)TReadyMinFwdRetry @F @T @F @F @T @T @TL(2)
fbCheckReady.bReady

@RT(7)Trans49 @F
@Step @RT(13)S_MinFwdRetry @F @F @F @F @RT(0) @F
@AcbCont @RT(7)unnamed @F 3
@Acb @RT(20)AStartMovementFwdBwd @F @T @RT(1)P @RT(0) @F @F @T @TL(4)
bMoveBwdDone := FALSE;
miErrorNo := cIdentSpeedMinFwdStart;
aStartMovementBwd();

@F
@Acb @RT(28)ACheckActMovementFwdBwdReady @F @T @RT(1)N @RT(0) @F @F @T @TL(5)
fbCheckReady(DeviceId := evStartRequestData.DeviceId);
IF fbCheckReady.bReady THEN
   bMoveBwdDone := TRUE;
END_IF;

@F
@Acb @RT(19)AStopMovementFwdBwd @F @T @RT(2)P0 @RT(0) @F @F @T @TL(3)
aStopMovementBwd();

@F

@AltBranch @RT(3)alt @F 2
@TransSeq @RT(4)tseq @F 1
@Trans @RT(12)TMoveBwdDone @F @T @F @F @T @T @TL(2)
bMoveBwdDone

@RT(12)TMoveBwdDone @F

@TransSeq @RT(4)tseq @F 4
@Trans @RT(12)TStopMoveBwd @F @T @F @F @T @F @TL(6)
sv_GlobalIdentMinSpeedStatus.Status = tnCalibState_Aborted OR
sv_GlobalIdentMinSpeedStatus.Status = tnCalibState_None
OR sv_iPendingAlarms <> 0
OR mActMovement^.bRedo = FALSE

@RT(12)TStopMoveBwd @F
@Step @RT(13)S_StopMoveBwd @F @F @T @F @RT(0) @F
@AcbCont @RT(7)unnamed @F 1
@Acb @RT(20)AStopMoveErrorBwdFwd @F @T @RT(1)P @RT(0) @F @F @T @TL(2)
aStopMovementError(sMovementName := CONCAT(sMoveName, ' min ident Fwd: Bwd to start position'));

@F

@Trans @RT(7)TReset2 @F @T @F @F @T @T @TL(2)
TRUE

@RT(7)TReset2 @F
@Goto @RT(7)S_RESET @F @F

@Step @RT(23)S_CHECK_ALARMS_RETRYFWD @F @F @F @F @RT(0) @F
@AcbCont @RT(7)unnamed @F 0

@AltBranch @RT(3)alt @F 2
@TransSeq @RT(4)tseq @F 1
@Trans @RT(9)TRetryFwd @F @T @F @F @T @T @TL(2)
S_CHECK_ALARMS_RETRYFWD.T > T#1s

@RT(9)TRetryFwd @F

@TransSeq @RT(4)tseq @F 2
@Trans @RT(14)TStopIdentFwd4 @F @T @F @F @T @F @TL(2)
sv_iPendingAlarms <> 0

@RT(14)TStopIdentFwd4 @F
@Goto @RT(13)S_StopMoveBwd @F @F

@Goto @RT(11)S_CALIB_FWD @F @F

@Step @RT(25)S_InitStartMovementBwdFwd @F @F @F @F @RT(0) @F
@AcbCont @RT(7)unnamed @F 3
@Acb @RT(24)AInitStartMovementBwdFwd @F @T @RT(1)P @RT(0) @F @F @T @TL(4)
bMoveFwdDone := FALSE;
miErrorNo := cIdentSpeedMinFwdInit;
aStartMovementFwd();

@F
@Acb @RT(29)ACheckInitMovementBwdFwdReady @F @T @RT(1)N @RT(0) @F @F @T @TL(5)
fbCheckReady(DeviceId := evStartRequestData.DeviceId);
IF fbCheckReady.bReady THEN
   bMoveFwdDone := TRUE;
END_IF;

@F
@Acb @RT(23)AStopInitMovementBwdFwd @F @T @RT(2)P0 @RT(0) @F @F @T @TL(2)
aStopMovementFwd();

@F

@AltBranch @RT(3)alt @F 2
@TransSeq @RT(4)tseq @F 1
@Trans @RT(7)Trans35 @F @T @F @F @T @T @TL(2)
bMoveFwdDone

@RT(7)Trans35 @F

@TransSeq @RT(4)tseq @F 4
@Trans @RT(16)TStopInitMoveFwd @F @T @F @F @T @F @TL(5)
sv_GlobalIdentMinSpeedStatus.Status = tnCalibState_Aborted OR
sv_GlobalIdentMinSpeedStatus.Status = tnCalibState_None
OR sv_iPendingAlarms <> 0
OR mActMovement^.bRedo = FALSE

@RT(16)TStopInitMoveFwd @F
@Step @RT(17)S_StopInitMoveFwd @F @F @T @F @RT(0) @F
@AcbCont @RT(7)unnamed @F 1
@Acb @RT(21)AStopMoveErrorInitFwd @F @T @RT(1)P @RT(0) @F @F @T @TL(2)
aStopMovementError(sMovementName := CONCAT(sMoveName, ' min ident Bwd: Fwd to initial position'));

@F

@Trans @RT(17)TResetInitMoveFwd @F @T @F @F @T @T @TL(2)
TRUE

@RT(17)TResetInitMoveFwd @F
@Goto @RT(7)S_RESET @F @F

@Step @RT(23)S_CHECK_ALARMS_STARTBWD @F @F @F @F @RT(0) @F
@AcbCont @RT(7)unnamed @F 0

@AltBranch @RT(3)alt @F 2
@TransSeq @RT(4)tseq @F 1
@Trans @RT(13)TStartInitBwd @F @T @F @F @T @T @TL(2)
S_CHECK_ALARMS_STARTBWD.T > T#100ms

@RT(13)TStartInitBwd @F

@TransSeq @RT(4)tseq @F 2
@Trans @RT(14)TStopIdentFwd3 @F @T @F @F @T @F @TL(2)
sv_iPendingAlarms <> 0

@RT(14)TStopIdentFwd3 @F
@Goto @RT(17)S_StopInitMoveFwd @F @F

@Step @RT(15)S_INITCALIB_BWD @F @F @F @F @RT(0) @F
@AcbCont @RT(7)unnamed @F 1
@Acb @RT(13)AInitCalibBwd @F @T @RT(1)P @RT(0) @F @F @T @TL(26)
iFileCounter := 1;
IF (CHECK_REF(mActMovement^.prSizeFactorBwd^)) THEN
   IF (mActMovement^.prSizeFactorBwd^ > 0.0) THEN
      rVelocitSizeFactor := mActMovement^.prSizeFactorBwd^;
   END_IF;
ELSE
   rVelocitSizeFactor := 1.0;
END_IF;
rRefSpeedLimit := 0.01 * mActMovement^.prVelocityLimitBwd^;
rMaxPressureLimit := mActMovement^.prMaxPressureBwd^;
IF CHECK_REF(mActMovement^.prMaxPressureBwdHydr^) THEN
   rMaxRefPressureLimit := mActMovement^.prMaxPressureBwdHydr^;
   IF (rMaxRefPressureLimit > 0.0) THEN
      rPressureFactorBwd := rMaxPressureLimit / rMaxRefPressureLimit;
   ELSE
      rPressureFactorBwd := 1.0;
   END_IF;
ELSE
   rMaxRefPressureLimit := mActMovement^.prMaxPressureFwd^;
   rPressureFactorBwd := 1.0;
END_IF;

aCalcMinSpeedOutput.bStart := TRUE;

dummy := Print('Calib min output %s Bwd started', sMoveName);

@F

@Trans @RT(13)TInitCalibBwd @F @T @F @F @T @T @TL(2)
S_INITCALIB_BWD.T>T#1s

@RT(13)TInitCalibBwd @F
@Step @RT(11)S_CALIB_BWD @F @F @T @F @RT(0) @F
@AcbCont @RT(7)unnamed @F 4
@Acb @RT(11)ADoCalibBwd @F @T @RT(1)P @RT(0) @F @F @T @TL(66)
mActMovement^.pConstBwdVis^.Velocity.Output.rOutputValue := rRefSpeedLimit * rVelocitSizeFactor;
mActMovement^.pConstBwdVis^.Velocity.rMinOutput := 0.0;
mActMovement^.pConstBwdVis^.Pressure.Output.rOutputValue := MAX(mActMovement^.pConstBwdVis^.Pressure.Output.rOutputValue, rMaxPressureLimit);
mActMovement^.pConstBwdVis^.Pressure.Output.rRamp := MAX(1.0e10, ConstVisBwd.Pressure.Output.rRamp);
IF mActMovement^.bPositionIncreasingFwd THEN
   mActMovement^.prIdentPosition^ := mActMovement^.prStroke^ * mrMinPositionFactor;
   mrMaxLimitPosition := rStartFactor * mActMovement^.prIdentPosition^ + (1.0 - rStartFactor) * mActMovement^.prPosition^;
   IF (mActMovement^.prPosition^ - mActMovement^.prIdentPosition^) > 0.0 THEN
      rMinStopRamp := rMinStrokeFactor * rRefSpeedLimit  * rRefSpeedLimit / ABS(mActMovement^.prIdentPosition^ - mActMovement^.prPosition^);
   ELSE
      rMinStopRamp := 0.0;
   END_IF;
   mActMovement^.prStopRamp^ := MAX(mActMovement^.pConstBwdVis^.Velocity.Output.rRamp, rMinStopRamp);
   mrMinLimitPosition := mActMovement^.prIdentPosition^ + 0.5 * rRefSpeedLimit  * rRefSpeedLimit / mActMovement^.prStopRamp^;
ELSE
   mActMovement^.prIdentPosition^ := mActMovement^.prStroke^ * mrMaxPositionFactor;
   mrMinLimitPosition := rStartFactor * mActMovement^.prPosition^ + (1.0 - rStartFactor) * mActMovement^.prIdentPosition^;
   IF (mActMovement^.prIdentPosition^ - mActMovement^.prPosition^) > 0.0 THEN
      rMinStopRamp := rMinStrokeFactor * rRefSpeedLimit  * rRefSpeedLimit / ABS(mActMovement^.prIdentPosition^ - mActMovement^.prPosition^);
   ELSE
      rMinStopRamp := 0.0;
   END_IF;
   mActMovement^.prStopRamp^ := MAX(mActMovement^.pConstBwdVis^.Velocity.Output.rRamp, rMinStopRamp);
   mrMaxLimitPosition := mActMovement^.prIdentPosition^ - 0.5 * rRefSpeedLimit  * rRefSpeedLimit / mActMovement^.prStopRamp^;
END_IF;
mActMovement^.pbMoveIdent^ := TRUE;

bMoveIdentDone := FALSE;

mrRefVelocity := rRefSpeedLimit;
mrRefPressure := rMaxRefPressureLimit;

aStartMeasurement();

bStopUnstable := FALSE;
bTimeOut := FALSE;
IF rRefSpeedLimit > 0.0 THEN
   rMoveStrokeTime := mActMovement^.prStroke^ / rRefSpeedLimit;
ELSE
   rMoveStrokeTime := 0.0;
END_IF;
dMaxMoveTime := T#5s + LINT_TO_TIME(REAL_TO_LINT(rMoveStrokeTime*1.0e6));
IF (dMaxMoveTime > dMoveTimeLimit) THEN
   dMaxMoveTime := dMoveTimeLimit;
   bMoveTimeLimited := TRUE;
   rStartPosition := mActMovement^.prPosition^;
   IF (mActMovement^.bPositionIncreasingFwd) THEN
      rMinMovementPosition := rStartPosition - 0.1 * (mrMaxLimitPosition - mrMinLimitPosition);
   ELSE;
      rMinMovementPosition := rStartPosition + 0.1 * (mrMaxLimitPosition - mrMinLimitPosition );
   END_IF;
ELSE
   bMoveTimeLimited := FALSE;
END_IF;

TimeOut(IN := FALSE,
        PT := dMaxMoveTime);
IF (mActMovement^.pdMaxMoveTimeBwd^ < dMaxMoveTime + dMoveTimeOffset) THEN
   mActMovement^.pdMaxMoveTimeBwd^ := dMaxMoveTime + dMoveTimeOffset;
END_IF;
mActMovement^.prVelocityBwd^ := rRefSpeedLimit;

sWriteSpeedLimit := REAL_TO_STRING(rRefSpeedLimit);
dummy := Print('Calib min output: act. min output: %s', sWriteSpeedLimit);
miErrorNo := cIdentSpeedMinBwdIdent;

@F
@Acb @RT(17)AStartMovementBwd @F @T @RT(1)P @RT(0) @F @F @T @TL(9)
evStartRequestData.DeviceId := mActMovement^.DeviceId;
evStartRequestData.MoveDir := cMoveBwd;
IF mActMovement^.MoveId > cMoveNone THEN
   evStartRequestData.MoveId := cMoveDecompAftPlast;
ELSE
   evStartRequestData.MoveId := cMoveBwd;
END_IF;
SET_EVENT(evStartRequest, evStartRequestData);

@F
@Acb @RT(25)ACheckActMovementBwdReady @F @T @RT(1)N @RT(0) @F @F @T @TL(28)
fbCheckReady(DeviceId := evStartRequestData.DeviceId);

TimeOut(IN :=TRUE);
IF fbCheckReady.bReady THEN
   aStopMeasurement();
   aStopMovementBwd();
   bMoveIdentDone := TRUE;
ELSIF TimeOut.Q THEN
   aStopMeasurement();
   aStopMovementBwd();
   IF (bMoveTimeLimited) AND
     ((mActMovement^.bPositionIncreasingFwd AND (mActMovement^.prPosition^ < rMinMovementPosition)) OR
      (NOT mActMovement^.bPositionIncreasingFwd AND (mActMovement^.prPosition^ > rMinMovementPosition))) THEN
      bMoveIdentDone := TRUE;
      dummy := Print('Calib min output: max move time reached with act. min output %s', sWriteSpeedLimit);
   ELSE
      bTimeOut := TRUE;
      dummy := Print('Calib min output: timeout with act. min output %s', sWriteSpeedLimit);
   END_IF;
ELSIF (abSpeedMeasure.aMeasure.bSpeedUnStable) THEN
   aStopMeasurement();
   aStopMovementBwd();
   bStopUnstable := TRUE;
   sWriteSpeedLimit := REAL_TO_STRING(rRefSpeedLimit);
   dummy := Print('Calib min output: unstable speed with act. min output %s', sWriteSpeedLimit);
END_IF;

@F
@Acb @RT(16)AStopMovementBwd @F @T @RT(2)P0 @RT(0) @F @F @T @TL(5)
mActMovement^.pConstBwdVis^ := ConstVisBwd;
mActMovement^.pdMaxMoveTimeBwd^ := dMaxMoveTimeSaveBwd;

TimeOut(IN := FALSE);

@F

@AltBranch @RT(3)alt @F 2
@TransSeq @RT(4)tseq @F 1
@Trans @RT(7)Trans14 @F @T @F @F @T @T @TL(4)
bMoveIdentDone OR
bTimeOut OR
bStopUnstable

@RT(7)Trans14 @F

@TransSeq @RT(4)tseq @F 4
@Trans @RT(13)TStopCalibBwd @F @T @F @F @T @F @TL(5)
sv_GlobalIdentMinSpeedStatus.Status = tnCalibState_Aborted OR
sv_GlobalIdentMinSpeedStatus.Status = tnCalibState_None
OR sv_iPendingAlarms <> 0
OR mActMovement^.bRedo = FALSE

@RT(13)TStopCalibBwd @F
@Step @RT(14)S_StopCalibBwd @F @F @T @F @RT(0) @F
@AcbCont @RT(7)unnamed @F 1
@Acb @RT(22)AStopMoveErrorCalibBwd @F @T @RT(1)P @RT(0) @F @F @T @TL(3)
aStopMovementBwd();
aStopMovementError(sMovementName := CONCAT(sMoveName, ' min ident Bwd'));

@F

@Trans @RT(14)TResetCalibBwd @F @T @F @F @T @F @TL(2)
TRUE

@RT(14)TResetCalibBwd @F
@Goto @RT(7)S_RESET @F @F

@Step @RT(18)S_CHECK_ALARMS_BWD @F @F @F @F @RT(0) @F
@AcbCont @RT(7)unnamed @F 0

@AltBranch @RT(3)alt @F 2
@TransSeq @RT(4)tseq @F 1
@Trans @RT(14)TStartWriteBwd @F @T @F @F @T @T @TL(2)
S_CHECK_ALARMS_BWD.T > T#100ms

@RT(14)TStartWriteBwd @F

@TransSeq @RT(4)tseq @F 2
@Trans @RT(14)TStopIdentBwd2 @F @T @F @F @T @F @TL(2)
sv_iPendingAlarms <> 0

@RT(14)TStopCalibBwd2 @F
@Goto @RT(14)S_StopCalibBwd @F @F

@Step @RT(11)S_WRITE_BWD @F @F @F @F @RT(0) @F
@AcbCont @RT(7)unnamed @F 1
@Acb @RT(9)AWriteBwd @F @T @RT(1)P @RT(0) @F @F @T @TL(14)
abSpeedMeasure.aGetMaxValues(rMaxSpeed => mrMaxVelocity,
                             rMaxPressure => mrMaxPressure,
                             bPressureLimitReached => mbPressureLimitReached,
                             bSpeedLimitReached => mbVelocityLimitReached);
IF mbprActPressureLinked THEN
   rMaxPressureBwd := MAX(rMaxPressureBwd, mrMaxPressure);
   dummy := Print('Calib min output: with act. min output %s max pressure %f needed', sWriteSpeedLimit, mrMaxPressure);
END_IF;
sFileName := CONCAT(sMoveName,"_MINSPEED_BWD_");
aWriteLog(sFileName := sFileName,
          iFileCounter := iFileCounter,
          bDeleteFiles := TRUE);
iFileCounter := iFileCounter + 1;

@F

@Trans @RT(9)TWriteBwd @F @T @F @F @T @T @TL(2)
mbLogFileSaved

@RT(9)TWriteBwd @F
@Step @RT(20)S_CHECK_MINSPEED_BWD @F @F @F @F @RT(0) @F
@AcbCont @RT(7)unnamed @F 1
@Acb @RT(17)ACheckMinSpeedBwd @F @T @RT(1)P @RT(0) @F @F @T @TL(20)
aCalcMinSpeedOutput(rMaxSpeedLimit := mActMovement^.prVelocityLimitBwd^,
                    rActRefSpeed := rRefSpeedLimit,
                    rActMinSpeed := abSpeedMeasure.aGetMaxValues.rMaxSpeed,
                    bUnstable := abSpeedMeasure.aGetMaxValues.bSpeedLimitUnStable,
                    bTimeOut := bTimeOut);
bMinBwdDetected := aCalcMinSpeedOutput.bMinDetected;
IF (bMinBwdDetected) THEN
   rSpeedLimitBwd := aCalcMinSpeedOutput.rMinSpeed;
   dummy := Print('Calib min output %s Bwd finished: min output bwd = %f$N', sMoveName, rSpeedLimitBwd);
ELSE
   bMinBwdRetry := TRUE;
   rRefSpeedLimit := aCalcMinSpeedOutput.rRefSpeed;
   aCalcMinSpeedOutput.bStart := FALSE;
END_IF;

mActMovement^.pConstBwdVis^ := ConstVisBwd;
mActMovement^.prVelocityBwd^ := rSpeedLimitBwd;
mActMovement^.pdMaxMoveTimeBwd^ := dMaxMoveTimeSaveBwd;

@F

@AltBranch @RT(3)alt @F 2
@TransSeq @RT(4)tseq @F 1
@Trans @RT(15)TMaxBwdDetected @F @T @F @F @T @T @TL(2)
bMinBwdDetected

@RT(15)TMaxBwdDetected @F

@TransSeq @RT(4)tseq @F 8
@Trans @RT(12)TMaxBwdRetry @F @T @F @F @T @T @TL(2)
bMinBwdRetry

@RT(12)TMaxBwdRetry @F
@Step @RT(18)S_ReadyMinBwdRetry @F @F @F @F @RT(0) @F
@AcbCont @RT(7)unnamed @F 1
@Acb @RT(17)AReadyMinBwdRetry @F @T @RT(1)N @RT(0) @F @F @T @TL(2)
fbCheckReady(DeviceId := mActMovement^.DeviceId);

@F

@Trans @RT(17)TReadyMinBwdRetry @F @T @F @F @T @T @TL(2)
fbCheckReady.bReady

@RT(7)Trans49 @F
@Step @RT(13)S_MinBwdRetry @F @F @F @F @RT(0) @F
@AcbCont @RT(7)unnamed @F 3
@Acb @RT(20)AStartMovementBwdFwd @F @T @RT(1)P @RT(0) @F @F @T @TL(4)
bMoveFwdDone := FALSE;
miErrorNo := cIdentSpeedMinBwdStart;
aStartMovementFwd();

@F
@Acb @RT(28)ACheckActMovementBwdFwdReady @F @T @RT(1)N @RT(0) @F @F @T @TL(5)
fbCheckReady(DeviceId := evStartRequestData.DeviceId);
IF fbCheckReady.bReady THEN
   bMoveFwdDone := TRUE;
END_IF;

@F
@Acb @RT(19)AStopMovementBwdFwd @F @T @RT(2)P0 @RT(0) @F @F @T @TL(4)
aStopMovementFwd();

@F

@AltBranch @RT(3)alt @F 2
@TransSeq @RT(4)tseq @F 1
@Trans @RT(12)TMoveFwdDone @F @T @F @F @T @T @TL(2)
bMoveFwdDone

@RT(12)TMoveFwdDone @F

@TransSeq @RT(4)tseq @F 4
@Trans @RT(12)TStopMoveFwd @F @T @F @F @T @F @TL(6)
sv_GlobalIdentMinSpeedStatus.Status = tnCalibState_Aborted OR
sv_GlobalIdentMinSpeedStatus.Status = tnCalibState_None
OR sv_iPendingAlarms <> 0
OR mActMovement^.bRedo = FALSE

@RT(12)TStopMoveFwd @F
@Step @RT(13)S_StopMoveFwd @F @F @T @F @RT(0) @F
@AcbCont @RT(7)unnamed @F 1
@Acb @RT(17)AStopMoveErrorFwd @F @T @RT(1)P @RT(0) @F @F @T @TL(2)
aStopMovementError(sMovementName := CONCAT(sMoveName, ' min ident Bwd: Fwd to start position'));

@F

@Trans @RT(9)TResetBwd @F @T @F @F @T @T @TL(2)
TRUE

@RT(9)TResetBwd @F
@Goto @RT(7)S_RESET @F @F

@Step @RT(23)S_CHECK_ALARMS_RETRYBWD @F @F @F @F @RT(0) @F
@AcbCont @RT(7)unnamed @F 0

@AltBranch @RT(3)alt @F 2
@TransSeq @RT(4)tseq @F 1
@Trans @RT(9)TRetryBwd @F @T @F @F @T @T @TL(2)
S_CHECK_ALARMS_RETRYBWD.T > T#1s

@RT(9)TRetryBwd @F

@TransSeq @RT(4)tseq @F 2
@Trans @RT(14)TStopIdentBwd4 @F @T @F @F @T @F @TL(2)
sv_iPendingAlarms <> 0

@RT(14)TStopIdentBwd4 @F
@Goto @RT(13)S_StopMoveFwd @F @F

@Goto @RT(11)S_CALIB_BWD @F @F

@Step @RT(12)S_MoveEndBwd @F @F @F @F @RT(0) @F
@AcbCont @RT(7)unnamed @F 3
@Acb @RT(11)AMoveEndBwd @F @T @RT(1)P @RT(0) @F @F @T @TL(23)
bMoveBwdDone := FALSE;

IF mActMovement^.bPositionIncreasingFwd THEN
   mActMovement^.prIdentPosition^ := mrBwdStopPosition;
ELSE
   mActMovement^.prIdentPosition^ := mActMovement^.prStroke^ - mrBwdStopPosition;
END_IF;
mActMovement^.prStopRamp^ := 1.0e10;
mActMovement^.pConstBwdVis^.Pressure.Output.rRamp := MAX(1.0e20,mActMovement^.pConstBwdVis^.Pressure.Output.rRamp);
mActMovement^.pConstBwdVis^.Pressure.rMinOutput := 0.1 * rMaxPressureLimit;
mActMovement^.pbMoveIdent^ := TRUE;

evStartRequestData.DeviceId := mActMovement^.DeviceId;
evStartRequestData.MoveDir := cMoveBwd;
IF mActMovement^.MoveId > cMoveNone THEN
   evStartRequestData.MoveId := cMoveDecompAftPlast;
ELSE
   evStartRequestData.MoveId := cMoveBwd;
END_IF;
miErrorNo := cIdentSpeedMinEnd;
SET_EVENT(evStartRequest, evStartRequestData);

@F
@Acb @RT(21)ACheckMoveEndBwdReady @F @T @RT(1)N @RT(0) @F @F @T @TL(5)
fbCheckReady(DeviceId := evStartRequestData.DeviceId);
IF fbCheckReady.bReady THEN
   bMoveBwdDone := TRUE;
END_IF;

@F
@Acb @RT(16)AMoveEndBwdReady @F @T @RT(2)P0 @RT(0) @F @F @T @TL(2)
aStopMovementBwd();

@F

@AltBranch @RT(3)alt @F 2
@TransSeq @RT(4)tseq @F 1
@Trans @RT(15)TMoveEndBwdDone @F @T @F @F @T @T @TL(2)
bMoveBwdDone

@RT(15)TMoveEndBwdDone @F

@TransSeq @RT(4)tseq @F 4
@Trans @RT(15)TStopMoveEndBwd @F @T @F @F @T @F @TL(4)
sv_GlobalIdentMinSpeedStatus.Status = tnCalibState_Aborted OR
sv_GlobalIdentMinSpeedStatus.Status = tnCalibState_None
OR sv_iPendingAlarms <> 0

@RT(15)TStopMoveEndBwd @F
@Step @RT(16)S_StopMoveEndBwd @F @F @F @F @RT(0) @F
@AcbCont @RT(7)unnamed @F 1
@Acb @RT(20)AStopMoveErrorEndBwd @F @T @RT(1)P @RT(0) @F @F @T @TL(2)
aStopMovementError(sMovementName := CONCAT(sMoveName, ' min ident: Bwd to end position'));

@F

@Trans @RT(16)TResetMoveEndBwd @F @T @F @F @T @F @TL(2)
TRUE

@RT(16)TResetMoveEndBwd @F
@Goto @RT(7)S_RESET @F @F

@Step @RT(6)S_Done @F @F @F @F @RT(0) @F
@AcbCont @RT(7)unnamed @F 1
@Acb @RT(5)ADone @F @T @RT(1)P @RT(0) @F @F @T @TL(16)
mActMovement^.Status := tnCalibState_Done;
sv_GlobalIdentMinSpeedStatus.Status := tnCalibState_Done;

mActMovement^.prVelocityFwd^ := rSpeedLimitFwd;
mActMovement^.prVelocityBwd^ := rSpeedLimitBwd;
IF mbprActPressureLinked THEN
   IF CHECK_REF(mActMovement^.prIdentPressureFwd^) THEN
      aRound(rActNumber := rMaxPressureFwd, rStep := rPressureStep);
      mActMovement^.prIdentPressureFwd^ := MAX(mActMovement^.prIdentPressureFwd^, aRound.rRoundedNumber * rPressureFactorFwd);
   END_IF;
   IF CHECK_REF(mActMovement^.prIdentPressureBwd^) THEN
      aRound(rActNumber := rMaxPressureBwd, rStep := rPressureStep);
      mActMovement^.prIdentPressureBwd^ := MAX(mActMovement^.prIdentPressureBwd^, aRound.rRoundedNumber * rPressureFactorBwd);
   END_IF;
END_IF;

@F

@Trans @RT(5)TDone @F @T @F @F @T @T @TL(2)
TRUE

@RT(5)TDone @F
@Goto @RT(7)S_RESET @F @F
@END_SfcData
@SaActions 0
@SaTrans 0
@SaExits 0
@END_SfcBody

@@@BEG_Comment@@@
@TL(0)

@@@END_Comment@@@

@BEG_Body
@TL(35)
//stop all calibrations
// TEST
IF sv_GlobalIdentMinSpeedStatus.Command = tnCalibCommand_Stop THEN
    sv_GlobalIdentMinSpeedStatus.bStart := FALSE;
END_IF;
//
IF sv_GlobalIdentMinSpeedStatus.Command = tnCalibCommand_Stop OR (NOT sv_GlobalIdentMinSpeedStatus.bStart) THEN
    FOR i:= 1 TO cCalibMovements DO
        IF CHECK_REF(sv_GlobalIdentMinSpeedStatus.pMovements[i]^) THEN
            IF sv_GlobalIdentMinSpeedStatus.pMovements[i]^.Status = tnCalibState_Running OR
               sv_GlobalIdentMinSpeedStatus.pMovements[i]^.bRedo THEN
                sv_GlobalIdentMinSpeedStatus.pMovements[i]^.Status := tnCalibState_Aborted;
                sv_GlobalIdentMinSpeedStatus.pMovements[i]^.bRedo := FALSE;//FIXME: check if needed
                sv_GlobalIdentMinSpeedStatus.Status := tnCalibState_Aborted;
                EXIT;
            END_IF;
        END_IF;
    END_FOR;
    IF (sv_GlobalIdentMinSpeedStatus.Command = tnCalibCommand_Stop) THEN
       IF (sv_GlobalIdentMinSpeedStatus.Status <> tnCalibState_Aborted) THEN
          sv_GlobalIdentMinSpeedStatus.Status := tnCalibState_None;
       END_IF;

    END_IF;
ELSIF (sv_GlobalIdentMinSpeedStatus.Command = tnCalibCommand_Start) OR (sv_GlobalIdentMinSpeedStatus.bStart) THEN
    IF sv_OperationMode = nSetup THEN
        mbUseSingleMovement := FALSE;
        START_PROCESS_ALGORITHM(paMinCalibSequence);
    ELSE
        sv_GlobalIdentMinSpeedStatus.bStart := FALSE;
        SET_ALARM(erSetupModeRequiredForCalib);
    END_IF;
END_IF;
sv_GlobalIdentMinSpeedStatus.Command := tnCalibCommand_None;

@END_Body

@@@BEG_Comment@@@
@TL(0)

@@@END_Comment@@@

@BEG_SfcBody
18 18 17

@BEG_SfcData 2
@StepSeq @RT(4)sseq @F 15
@Step @RT(7)S_RESET @F @F @T @F @RT(0) @F
@AcbCont @RT(7)unnamed @F 3
@Acb @RT(6)AReset @F @T @RT(1)P @RT(0) @F @F @T @TL(2)
sv_bAutoIdentRunning := FALSE;

@F
@Acb @RT(14)AStopMovements @F @T @RT(1)N @RT(0) @F @F @T @TL(12)
(* stop all identification movements *)
FOR i:= 1 TO cCalibMovements DO
    IF CHECK_REF(sv_GlobalIdentMinSpeedStatus.pMovements[i]^) THEN
        IF sv_GlobalIdentMinSpeedStatus.pMovements[i]^.Status = tnCalibState_Running OR
           sv_GlobalIdentMinSpeedStatus.pMovements[i]^.bRedo THEN
            sv_GlobalIdentMinSpeedStatus.pMovements[i]^.Status := tnCalibState_Aborted;
            sv_GlobalIdentMinSpeedStatus.pMovements[i]^.bRedo := FALSE;//FIXME: check if needed
            EXIT;
        END_IF;
    END_IF;
END_FOR;

@F
@Acb @RT(9)AStopSelf @F @T @RT(1)P @RT(0) @F @F @T @TL(3)
sv_GlobalIdentMinSpeedStatus.bStart := FALSE;
STOP_PROCESS_ALGORITHM();

@F

@Trans @RT(7)Trans50 @F @T @F @F @T @T @TL(2)
TRUE

@RT(7)Trans50 @F
@Step @RT(6)S_INIT @F @T @F @F @RT(0) @F
@AcbCont @RT(7)unnamed @F 2
@Acb @RT(11)ASortCalibs @F @T @RT(1)P @RT(0) @F @F @T @TL(24)
sv_GlobalIdentMinSpeedStatus.Status := tnCalibState_Running;
miErrorNo := 0;

tmpMovements := sv_GlobalIdentMinSpeedStatus.pMovements;

(* get number of movements *)
FOR i:= 1 TO cCalibMovements DO
    IF NOT CHECK_REF(tmpMovements[i]^)  THEN
        EXIT;
    END_IF;
END_FOR;
iMaxMovements := i -1;

(* sort them by iOrder *)
FOR i := 1 TO iMaxMovements -1 DO
    FOR j := 1 TO iMaxMovements - 1 - i +1 DO
        IF tmpMovements[j]^.iOrder > tmpMovements[j + 1]^.iOrder THEN
            tmpM := tmpMovements[j];
            tmpMovements[j] := tmpMovements[j + 1];
            tmpMovements[j + 1] := tmpM;
        END_IF;
    END_FOR;
END_FOR;

@F
@Acb @RT(9)Action108 @F @T @RT(1)P @RT(0) @F @F @T @TL(3)
mCalibCounter := 0;
sv_GlobalIdentMinSpeedStatus.iCurrentStep := mCalibCounter;

@F

@AltBranch @RT(3)alt @F 2
@TransSeq @RT(4)tseq @F 1
@Trans @RT(7)Trans80 @F @T @F @F @T @T @TL(3)
NOT sv_bCoresActive AND
sv_iPendingAlarms = 0

@RT(7)Trans80 @T @TL(5)
Comment : Start with moving ejector and
mold in backward position, check if any failure
occured.
After that start the calibration cycle, if no alarm is
pending

@TransSeq @RT(4)tseq @F 4
@Trans @RT(7)Trans87 @F @T @F @F @T @F @TL(4)
sv_bCoresActive OR
sv_iPendingAlarms > 0

@RT(7)Trans87 @F
@Step @RT(6)Step74 @F @F @F @F @RT(0) @F
@AcbCont @RT(7)unnamed @F 1
@Acb @RT(14)AAnyCoreActive @F @F @RT(1)N @RT(0) @F @F @F @F

@Trans @RT(7)Trans88 @F @T @F @F @T @T @TL(3)
TRUE

@RT(7)Trans88 @F
@Goto @RT(7)S_RESET @F @F

@Step @RT(6)Step19 @F @F @F @F @RT(0) @F
@AcbCont @RT(7)unnamed @F 1
@Acb @RT(12)ASignalStart @F @T @RT(1)P @RT(0) @F @F @T @TL(2)
sv_bAutoIdentRunning := TRUE;

@F

@Trans @RT(7)Trans18 @F @T @F @F @T @T @TL(2)
TRUE

@RT(7)Trans18 @F
@Step @RT(17)S_MoveEjectorBack @F @F @F @F @RT(0) @F
@AcbCont @RT(7)unnamed @F 3
@Acb @RT(12)AEjectorBack @F @F @RT(1)P @RT(0) @F @F @F @F
@Acb @RT(9)Action116 @F @T @RT(1)N @RT(0) @F @F @T @TL(2)
fbCheckReady(DeviceId := DeviceIdEjector)

@F
@Acb @RT(17)AResetEjectorBack @F @T @RT(2)P0 @RT(0) @F @F @T @TL(7)
miErrorNo := 0;
sv_EjectorIdentMinMovement.prIdentPosition^ := 0.0;
sv_EjectorIdentMinMovement.prStopRamp^ := 0.0;
sv_EjectorIdentMinMovement.pbMoveIdent^ := FALSE;
sv_EjectorIdentMinMovement.pConstBwdVis^ := ConstBwdVis;

@F

@AltBranch @RT(3)alt @F 2
@TransSeq @RT(4)tseq @F 1
@Trans @RT(7)Trans72 @F @T @F @F @T @T @TL(3)
fbCheckReady.bReady AND
sv_iPendingAlarms = 0

@RT(7)Trans72 @F

@TransSeq @RT(4)tseq @F 4
@Trans @RT(7)Trans83 @F @T @F @F @T @F @TL(4)
sv_GlobalIdentMinSpeedStatus.Status = tnCalibState_Aborted OR
sv_GlobalIdentMinSpeedStatus.Status = tnCalibState_None
OR sv_iPendingAlarms <> 0

@RT(7)Trans83 @F
@Step @RT(13)S_StopEjector @F @F @F @F @RT(0) @F
@AcbCont @RT(7)unnamed @F 1
@Acb @RT(16)AStopEjeMovement @F @F @RT(1)P @RT(0) @F @F @F @F

@Trans @RT(7)Trans84 @F @T @F @F @T @T @TL(3)
TRUE

@RT(7)Trans84 @F
@Goto @RT(7)S_RESET @F @F

@Step @RT(14)S_MoveMoldBack @F @F @F @F @RT(0) @F
@AcbCont @RT(7)unnamed @F 3
@Acb @RT(9)AMoldBack @F @F @RT(1)P @RT(0) @F @F @F @F
@Acb @RT(9)Action118 @F @T @RT(1)N @RT(0) @F @F @T @TL(2)
fbCheckReady(DeviceId := DeviceIdMold)

@F
@Acb @RT(14)AResetMoldBack @F @T @RT(2)P0 @RT(0) @F @F @T @TL(7)
miErrorNo := 0;
sv_MoldIdentMinMovement.prIdentPosition^ := 0.0;
sv_MoldIdentMinMovement.prStopRamp^ := 0.0;
sv_MoldIdentMinMovement.pbMoveIdent^ := FALSE;
sv_MoldIdentMinMovement.pConstBwdVis^ := ConstBwdVis;

@F

@AltBranch @RT(3)alt @F 2
@TransSeq @RT(4)tseq @F 1
@Trans @RT(7)Trans81 @F @T @F @F @T @T @TL(3)
fbCheckReady.bReady AND
sv_iPendingAlarms = 0

@RT(7)Trans81 @F

@TransSeq @RT(4)tseq @F 4
@Trans @RT(7)Trans85 @F @T @F @F @T @F @TL(4)
sv_GlobalIdentMinSpeedStatus.Status = tnCalibState_Aborted OR
sv_GlobalIdentMinSpeedStatus.Status = tnCalibState_None
OR sv_iPendingAlarms <> 0

@RT(7)Trans85 @F
@Step @RT(10)S_StopMold @F @F @F @F @RT(0) @F
@AcbCont @RT(7)unnamed @F 1
@Acb @RT(17)AStopMoldMovement @F @F @RT(1)P @RT(0) @F @F @F @F

@Trans @RT(7)Trans86 @F @T @F @F @T @T @TL(2)
TRUE

@RT(7)Trans86 @F
@Goto @RT(7)S_RESET @F @F

@Step @RT(14)S_CALIB_SINGLE @F @F @T @F @RT(0) @F
@AcbCont @RT(7)unnamed @F 1
@Acb @RT(19)AStartMovementStart @F @T @RT(1)P @RT(0) @F @F @T @TL(5)
IF mCalibCounter < iMaxMovements THEN
   mCalibCounter := mCalibCounter +1;
   tmpMovements[mCalibCounter]^.bRedo := TRUE;
END_IF;

@F

@AltBranch @RT(3)alt @F 2
@TransSeq @RT(4)tseq @F 1
@Trans @RT(18)TCheckActMoveReady @F @T @F @F @T @T @TL(4)
tmpMovements[mCalibCounter]^.bRedo = FALSE AND
NOT(sv_GlobalIdentMinSpeedStatus.Status = tnCalibState_Aborted OR
    sv_GlobalIdentMinSpeedStatus.Status = tnCalibState_Error)

@RT(18)TCheckActMoveReady @F

@TransSeq @RT(4)tseq @F 2
@Trans @RT(11)TCheckError @F @T @F @F @T @F @TL(4)
sv_GlobalIdentMinSpeedStatus.Status = tnCalibState_Aborted OR
sv_GlobalIdentMinSpeedStatus.Status = tnCalibState_Error OR
iMaxMovements = 0

@RT(11)TCheckError @F
@Goto @RT(7)S_RESET @F @F

@Step @RT(11)S_CHECKNEXT @F @F @F @F @RT(0) @F
@AcbCont @RT(7)unnamed @F 0

@AltBranch @RT(3)alt @F 2
@TransSeq @RT(4)tseq @F 1
@Trans @RT(9)TNextUnit @F @T @F @F @T @T @TL(3)
mCalibCounter < iMaxMovements
//AND S_CHECKNEXT.T>T#3s

@RT(9)TNextUnit @F

@TransSeq @RT(4)tseq @F 4
@Trans @RT(10)TStopIdent @F @T @F @F @T @T @TL(2)
mCalibCounter >= iMaxMovements

@RT(10)TStopIdent @F
@Step @RT(11)S_StopIdent @F @F @F @F @RT(0) @F
@AcbCont @RT(7)unnamed @F 1
@Acb @RT(10)AStopIdent @F @T @RT(1)P @RT(0) @F @F @T @TL(2)
sv_GlobalIdentMinSpeedStatus.Status := tnCalibState_Done;

@F

@Trans @RT(6)TReset @F @T @F @F @T @T @TL(2)
TRUE

@RT(6)TReset @F
@Goto @RT(7)S_RESET @F @F

@Goto @RT(14)S_CALIB_SINGLE @F @F
@END_SfcData
@SaActions 5
@SaText @RT(12)AEjectorBack 1 @TL(20)
miErrorNo := cIdentSpeedMinSequence;

IF sv_EjectorIdentMinMovement.bPositionIncreasingFwd THEN
   sv_EjectorIdentMinMovement.prIdentPosition^ := mrBwdStopPosition;
ELSE
   sv_EjectorIdentMinMovement.prIdentPosition^ := sv_EjectorIdentMinMovement.prStroke^ - mrBwdStopPosition;
END_IF;
sv_EjectorIdentMinMovement.prStopRamp^ := 1.0e10;
ConstBwdVis := sv_EjectorIdentMinMovement.pConstBwdVis^;
sv_EjectorIdentMinMovement.pConstBwdVis^.Pressure.Output.rRamp := MAX(1.0e10, sv_EjectorIdentMinMovement.pConstBwdVis^.Pressure.Output.rRamp);
sv_EjectorIdentMinMovement.pConstBwdVis^.Pressure.rMinOutput := 0.1 * sv_EjectorIdentMinMovement.prMaxPressureBwd^;
sv_EjectorIdentMinMovement.pbMoveIdent^ := TRUE;

evStartRequestData.DeviceId := DeviceIdEjector;
evStartRequestData.MoveDir := cMoveBwd;
evStartRequestData.MoveId := cMoveBwd;
SET_EVENT(evStartRequest, evStartRequestData);

@SaText @RT(9)AMoldBack 1 @TL(19)
miErrorNo := cIdentSpeedMinSequence;

IF sv_MoldIdentMinMovement.bPositionIncreasingFwd THEN
   sv_MoldIdentMinMovement.prIdentPosition^ := mrBwdStopPosition;
ELSE
   sv_MoldIdentMinMovement.prIdentPosition^ := sv_MoldIdentMinMovement.prStroke^ - mrBwdStopPosition;
END_IF;
sv_MoldIdentMinMovement.prStopRamp^ := 1.0e10;
ConstBwdVis := sv_MoldIdentMinMovement.pConstBwdVis^;
sv_MoldIdentMinMovement.pConstBwdVis^.Pressure.Output.rRamp := MAX(1.0e10, sv_MoldIdentMinMovement.pConstBwdVis^.Pressure.Output.rRamp);
sv_MoldIdentMinMovement.pConstBwdVis^.Pressure.rMinOutput := 0.1 * sv_MoldIdentMinMovement.prMaxPressureBwd^;
sv_MoldIdentMinMovement.pbMoveIdent^ := TRUE;

evStartRequestData.DeviceId := DeviceIdMold;
evStartRequestData.MoveDir := cMoveBwd;
evStartRequestData.MoveId := cMoveBwd;
SET_EVENT(evStartRequest, evStartRequestData);

@SaText @RT(16)AStopEjeMovement 1 @TL(10)
evStopRequestData.DeviceId := DeviceIdEjector;
evStopRequestData.MoveDir := cMoveBwd;
evStopRequestData.MoveId := cMoveBwd;
SET_EVENT(evStopRequest, evStopRequestData);
IF sv_GlobalIdentMinSpeedStatus.Status <> tnCalibState_None THEN
    sv_GlobalIdentMinSpeedStatus.Status := tnCalibState_Aborted;
END_IF;

@SaText @RT(17)AStopMoldMovement 1 @TL(10)
evStopRequestData.DeviceId := DeviceIdMold;
evStopRequestData.MoveDir := cMoveBwd;
evStopRequestData.MoveId := cMoveBwd;
SET_EVENT(evStopRequest, evStopRequestData);
IF sv_GlobalIdentMinSpeedStatus.Status <> tnCalibState_None THEN
    sv_GlobalIdentMinSpeedStatus.Status := tnCalibState_Aborted;
END_IF;

@SaText @RT(14)AAnyCoreActive 1 @TL(6)
IF sv_bCoresActive THEN
   SET_ALARM(erCalibCoresActive);
END_IF;
sv_GlobalIdentMinSpeedStatus.Status := tnCalibState_Aborted;

@SaTrans 0
@SaExits 1
@SaExit @SaText @RT(14)E_NotSetupMode 1 @TL(2)
sv_OperationMode <> nSetup

@RT(7)S_RESET @RT(1)1 @F @F @SaSfc @RT(14)E_NotSetupMode 5 @RT(5)DUMMY
@BEG_SfcData 2
@ExitSeq @RT(4)sseq @F 3
@Step @RT(8)unnamed1 @F @T @F @F @RT(0) @F
@AcbCont @RT(7)unnamed @F 0

@Trans @RT(8)unnamed3 @F @T @F @F @T @T @TL(2)

@RT(8)unnamed3 @F
@Goto @RT(9)unlabeled @F @F
@END_SfcData

@END_SfcBody

@@@BEG_Comment@@@
@TL(2)
Coordinate sequential start of auto calib cycle
starts one auto calib movement after the other
@@@END_Comment@@@

@BEG_Body
@TL(27)
(**************************************** WARNING ********************************************
 *** The KEBA Kemro K2 System including software is not intended for safety control tasks! ***
 ***                       For further information see Comment tab!                        ***
 *********************************************************************************************)

//reset calib state after loading machine data

IF sv_DataState = nReadMachineData THEN
   //loading of machinedata in progress
   bMDLoadingInProgress := TRUE;
   RETURN;
END_IF;

IF sv_DataState = nReady AND bMDLoadingInProgress THEN
   FOR i := 1 TO sv_GlobalIdentMaxSpeedStatus.iMaxStep DO
      //set state to tnCalibState_None
      sv_GlobalIdentMaxSpeedStatus.pMovements[i]^.Status := tnCalibState_None;
   END_FOR;
   FOR i := 1 TO sv_GlobalIdentMinSpeedStatus.iMaxStep DO
      //set state to tnCalibState_None
      sv_GlobalIdentMinSpeedStatus.pMovements[i]^.Status := tnCalibState_None;
   END_FOR;
   bMDLoadingInProgress := FALSE;
END_IF;

@END_Body

@@@BEG_Comment@@@
@TL(0)

@@@END_Comment@@@
@END_Body

@END_Contents
